{attribute 'GeneratedUsingTerminal: EL4004-0000-0016'}
{attribute addProperty BoxType "EL4004-0000-0016"}
{attribute addProperty Description "EL4004 4Ch. Ana. Output 0-10V, 12bit"}
{attribute addProperty Physics "KK"}
{attribute addProperty Id "AO_Outputs_Channel_1AT %Q*AO_Output_Channel_BA7EBB7C2AO_Outputs_Channel_2AT %Q*AO_Output_Channel_BA7EBB7C2AO_Outputs_Channel_3AT %Q*AO_Output_Channel_BA7EBB7C2AO_Outputs_Channel_4AT %Q*AO_Output_Channel_BA7EBB7C2WcStateAT %I*WcState_0B2B16F91InfoDataAT %I*InfoData_32EB74EA10"}
{attribute addProperty CRC "2878501134"}
{attribute addProperty Size "19"}
TYPE EL4004_AB92710E EXTENDS EtcSlaveTerminalBase_947E5A46 :
STRUCT
	{attribute addProperty Name "AO_Outputs_Channel_1"}
	AO_Outputs_Channel_1 : AO_Output_Channel_BA7EBB7C;
	{attribute addProperty Name "AO_Outputs_Channel_2"}
	AO_Outputs_Channel_2 : AO_Output_Channel_BA7EBB7C;
	{attribute addProperty Name "AO_Outputs_Channel_3"}
	AO_Outputs_Channel_3 : AO_Output_Channel_BA7EBB7C;
	{attribute addProperty Name "AO_Outputs_Channel_4"}
	AO_Outputs_Channel_4 : AO_Output_Channel_BA7EBB7C;
	{attribute addProperty Name "WcState"}
	WcState : WcState_0B2B16F9;
	{attribute addProperty Name "InfoData"}
	InfoData : InfoData_32EB74EA;
END_STRUCT
END_TYPE

(* stored: Version 1.2.0.0, ProductVersion 3.1.4024.9
   DUT EL4004_AB92710E: Id {a96fe896-8ca9-4c13-bf86-120a65bf140b} *)
